// TIA Portal project "Tankfuellanlage_111" (V14)

(* hardware
DEVICE "S7-1200-Station_1"  S7-1200 Station
   slot 0: "Baugruppenträger_0"  S7-1200 Rack  Rack  V1.0
   slot 1: "PLC_1"  CPU 1214C DC/DC/DC  6ES7 214-1AG40-0XB0  V4.2
   slot 3: "AQ 1x12BIT_1"  AQ1 signal board  6ES7 232-4HA30-0XB0  V1.0
*)

// ===== PLC "PLC_1"  CPU 1214C DC/DC/DC =====

VAR_GLOBAL   // PLC tag table "Standard-Variablentabelle"
   "System_Byte" AT %MB100 : Byte;
   "FirstScan" AT %M100.0 : Bool;
   "DiagStatusUpdate" AT %M100.1 : Bool;
   "AlwaysTRUE" AT %M100.2 : Bool;
   "AlwaysFALSE" AT %M100.3 : Bool;
   "Clock_Byte" AT %MB110 : Byte;
   "Clock_10Hz" AT %M110.0 : Bool;
   "Clock_5Hz" AT %M110.1 : Bool;
   "Clock_2.5Hz" AT %M110.2 : Bool;
   "Clock_2Hz" AT %M110.3 : Bool;
   "Clock_1.25Hz" AT %M110.4 : Bool;
   "Clock_1Hz" AT %M110.5 : Bool;
   "Clock_0.625Hz" AT %M110.6 : Bool;
   "Clock_0.5Hz" AT %M110.7 : Bool;
   "B1" AT %I0.0 : Bool;   // Schwimmerschalter Tank 1 „Leer“
   "B2" AT %I0.1 : Bool;   // Schwimmerschalter Tank 1 „Voll“
   "B3" AT %I0.2 : Bool;   // Schwimmerschalter Tank 2 „Leer“
   "B4" AT %I0.3 : Bool;   // Schwimmerschalter Tank 2 „Voll“
   "B5" AT %I0.4 : Bool;   // Schwimmerschalter Tank 3 „Leer“
   "B6" AT %I0.5 : Bool;   // Schwimmerschalter Tank 3 „Voll“
   "Q1" AT %Q0.0 : Bool;   // Ventil für Tank 1
   "Q2" AT %Q0.1 : Bool;   // Ventil für Tank 2
   "Q3" AT %Q0.2 : Bool;   // Ventil für Tank 3
   "P1" AT %Q0.3 : Bool;   // Störung
   "AlleAusgänge" AT %QW0 : Word;
END_VAR

FUNCTION "fc_Tankfuellanlage" : Void   // FC1, SCL
{ S7_Optimized_Access := 'TRUE' }
VERSION : 0.1
BEGIN
   IF NOT "B1" THEN
       "Q1" := TRUE;
   END_IF;

   IF "Q1" AND "B2" THEN
       "Q1" := false;
   END_IF;

   IF NOT "B3" THEN
       "Q2" := TRUE;
   END_IF;

   IF "Q2" AND "B4" THEN
       "Q2" := false;
   END_IF;

   IF NOT "B5" THEN
       "Q3" := TRUE;
   END_IF;

   IF "Q3" AND "B6" THEN
       "Q3" := false;
   END_IF;
END_FUNCTION

ORGANIZATION_BLOCK "Main"   // OB1, LAD, ProgramCycle
TITLE = "Main Program Sweep (Cycle)"
{ S7_Optimized_Access := 'TRUE' }
VERSION : 0.1
   VAR_INPUT
      Initial_Call : Bool;   // Initial call of this OB
      Remanence : Bool;   // =True, if remanent data are available
   END_VAR
BEGIN

REGION Network 1
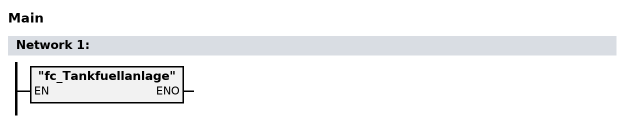
   RUNG wire#powerrail
      "fc_Tankfuellanlage"()
   END_RUNG
   // the same network as SCL:
   "fc_Tankfuellanlage"();
END_REGION
END_ORGANIZATION_BLOCK

ORGANIZATION_BLOCK "Startup"   // OB100, SCL, Startup
TITLE = "Complete Restart"
{ S7_Optimized_Access := 'TRUE' }
VERSION : 0.1
   VAR_INPUT
      LostRetentive : Bool;   // True if retentive data are lost
      LostRTC : Bool;   // True if date and time are lost
   END_VAR
BEGIN
   "AlleAusgänge"
END_ORGANIZATION_BLOCK